TYPE ST_UnloadingBottleParams :
STRUCT
END_STRUCT
END_TYPE

(* stored: Version 1.1.0.1, ProductVersion 3.1.4024.15
   DUT ST_UnloadingBottleParams: Id {e64e414a-1e76-43e8-8cbf-f40aa4daed91} *)
